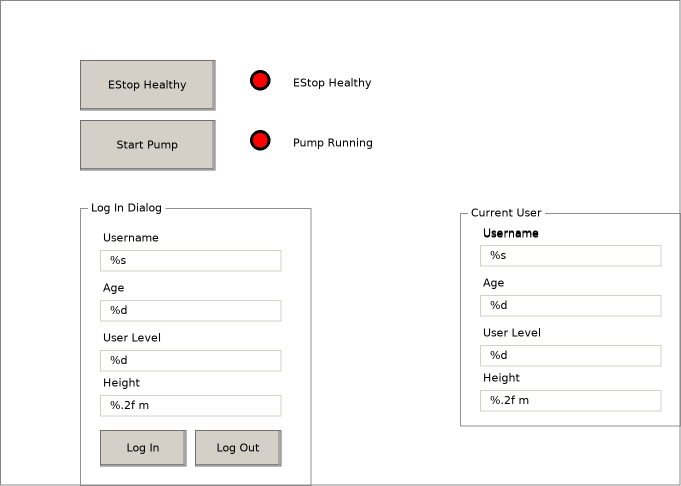
VISUALIZATION Visualization  // 681x486
    Button (80,60 135x50), "EStop Healthy"
        toggle DigitalInputs.EStopHealthy
    Button (80,120 135x50), "Start Pump"
        tap DigitalInputs.StartPumpPb
    Ellipse (250,130 20x20), colour toggle: DigitalOutputs.HydraulicPumpRunningLamp
    Label (290,135 151x16), "Pump Running"
    Ellipse (250,70 20x20), colour toggle: DigitalInputs.EStopHealthy
    Label (290,75 151x16), "EStop Healthy"
    GroupBox (80,200 231x286), "Log In Dialog"
        Textfield (20,50 181x21), "%s", text variable: Objects.HmiInterface.UserName
            OnMouseClick: write the text variable via Default
        Label (20,80 151x16), "Age"
        Textfield (20,100 181x21), "%d", text variable: Objects.HmiInterface.UserAge
            OnMouseClick: write the text variable via Default
        Label (20,130 151x16), "User Level"
        Textfield (20,150 181x21), "%d", text variable: Objects.HmiInterface.UserLevel
            OnMouseClick: write the text variable via Default
        Label (20,175 151x16), "Height"
        Textfield (20,195 181x21), "%.2f m", text variable: Objects.HmiInterface.UserHeight
            OnMouseClick: write the text variable via Default
        Button (20,230 86x36), "Log In"
            tap Objects.HmiInterface.LogIn
        Button (115,230 86x36), "Log Out"
            tap Objects.HmiInterface.LogOut
        Label (400,25 151x16), "Username"
        Label (20,30 151x16), "Username"
    GroupBox (460,205 221x221), "Current User"
        Label (20,21 151x16), "Username"
    Textfield (480,245 181x21), "%s", text variable: Globals.CurrentUserName
    Label (480,275 151x16), "Age"
    Textfield (480,295 181x21), "%d", text variable: Globals.CurrentUserAge
    Label (480,325 151x16), "User Level"
    Textfield (480,345 181x21), "%d", text variable: Globals.CurrentUserLevel
    Label (480,370 151x16), "Height"
    Textfield (480,390 181x21), "%.2f m", text variable: Globals.CurrentUserHeight
END_VISUALIZATION

(* stored: Version 1.1.0.1, ProductVersion 3.1.4024.9
   Visu Visualization: Id {c1b85e8b-8590-0739-2bb2-2c9dea61dce1} *)
